// TIA Portal V20 export
DATA_BLOCK "DB_NordSetPoint"   // DB33
// stored: Access Published, MemoryReserve 100, Namespace Global
   VAR
      Line : Struct
         ProductionLine : Struct   // -(0 - 16000) -> (CW: 0 - 100%) || +(0 - 16000) (CCW: 0 - 100%) || freq. has been set via NORDCON
            Conveyor : Array[_.gminProductionLine.._.gmaxProductionLine] of DInt;
         END_STRUCT;
         EmptyLine : Struct   // -(0 - 16000) -> (CW: 0 - 100%) || +(0 - 16000) (CCW: 0 - 100%) || freq. has been set via NORDCON
            Conveyor : Array[_.gminEmptyLine.._.gmaxEmptyLine] of DInt;
         END_STRUCT;
         PackedLine : Struct   // -(0 - 16000) -> (CW: 0 - 100%) || +(0 - 16000) (CCW: 0 - 100%) || freq. has been set via NORDCON
            Conveyor : Array[_.gminPackedLine.._.gmaxPackedLine] of DInt;
         END_STRUCT;
      END_STRUCT;
   END_VAR
BEGIN
END_DATA_BLOCK
